// TwinCAT 3 PLC project kallebol_PLC_proj
// ProgramVersion: 3.1.4024.0
// libraries:
//   Tc2_MC2, * (Beckhoff Automation GmbH)
//   Tc2_Standard, * (Beckhoff Automation GmbH)
//   Tc2_System, * (Beckhoff Automation GmbH)
//   Tc3_Module, * (Beckhoff Automation GmbH)
// project tree:
//   / PlcTask.TcTTO
//   POUs/ MAIN.TcPOU
//   POUs/POUs/ FB_Azimuth.TcPOU, FB_Elevation.TcPOU
// real-time tasks:
//   TASK PlcTask: cycle T#10ms, priority 20, ADS port 350
// motion (NC):
//   TASK Azimuth_NC_task SAF: cycle T#2ms, priority 4, ADS port 501
//   TASK Azimuth_NC_task SVB: cycle T#10ms, priority 8, ADS port 511
//   AXIS Axis 3 (id 3)
//     General: UnitName=°
//     Dynamic: Acceleration=15000, Deceleration=15000, Jerk=64125
//     Velo: RefSearch=142.5, RefSync=142.5, SlowManual=712.5, FastManual=4275, Fast=14250, Maximum=14250
//     PositionAreaControl: Enable=false
//     TargetPosControl: Enable=false
//     OtherSettings: AllowMotionCmdToSlave=true
//     encoder EncType=8
//       EncPara: ScaleFactorNumerator=360, ScaleFactorDenominator=1048576, MaxCount=#xffffffff, EncPositionSource=1
//     drive DrvType=9
//       DrvPara: MaxCount=#xffffffff, DriveControlDWord=#x00030100
//         Analog: VeloReferenz=15675, VeloScale=1.02400649589962, TorqueSetpointScale=10, ScaleFactorActTorque=0.1
//         TimeComp: TaskDelayCycles=1
//     controller CtrType=1
//       CtrPara: PriorControlFactor=1
//         PosDiffControl: Enable=false
//         Observer: BandWidth=20
// I/O:
//   DEVICE Device 1 (EtherCAT), AmsNetId 5.79.241.154.2.1
//     Term 1 (EK1200) [EK1200-5000 EtherCAT Power supply (2A E-Bus)]
//       Term 2 (EL7342) [EL7342 2Ch. DC motor output stage (50V, 3.5A)]
//       RS485_term [EL6021 Interface (RS422/485)]
//       Term 3 (EK1110) [EK1110 EtherCAT extension]
//     Drive 4 (AX5203-0000-0214) [AX5203-0000-0214 EtherCAT Drive (SoE, 2 Ch.)]
// variable links:
//   Azimuth_NC_task SAF/Axes/Axis 3 <-> Device 1 (EtherCAT)/Drive 4 (AX5203-0000-0214)
//     Drive/Inputs/In/nDataIn1 <-> AT 1/Following distance
//     Drive/Inputs/In/nDataIn3[0] <-> AT 1/Torque/force feedback value
//     Drive/Inputs/In/nDcOutputTime <-> InfoData/DcOutputShift
//     Drive/Inputs/In/nState1 <-> AT 1/Drive status word @bit 8
//     Drive/Inputs/In/nState2 <-> AT 1/Drive status word
//     Drive/Inputs/In/nState4 @bit 1 <-> WcState/InputToggle
//     Drive/Inputs/In/nState4 <-> WcState/WcState
//     Drive/Outputs/Out/nCtrl1 <-> MDT 1/Master control word @bit 8
//     Drive/Outputs/Out/nDataOut1 <-> MDT 1/Position command value
//     Enc/Inputs/In/nDataIn1 <-> AT 1/Position feedback 1 value
//     Enc/Inputs/In/nDcInputTime <-> InfoData/DcInputShift
//     Enc/Inputs/In/nState4 @bit 1 <-> WcState/InputToggle
//     Enc/Inputs/In/nState4 <-> WcState/WcState
//   kallebol_PLC_proj/kallebol_PLC_proj Instance <-> Device 1 (EtherCAT)/Term 1 (EK1200)/Term 2 (EL7342)
//     PlcTask Inputs/MAIN.Elevation.Encoder_Value <-> ENC Status Channel 1/Counter value
//     PlcTask Inputs/MAIN.Elevation.Error <-> DCM Status Channel 1/Status/Error
//     PlcTask Inputs/MAIN.Elevation.Homing_Switch <-> DCM Status Channel 1/Status/Digital input 1
//     PlcTask Inputs/MAIN.Elevation.Limit_Switch <-> DCM Status Channel 1/Status/Digital input 2
//     PlcTask Inputs/MAIN.Elevation.Moving_negative <-> DCM Status Channel 1/Status/Moving negative
//     PlcTask Inputs/MAIN.Elevation.Moving_positive <-> DCM Status Channel 1/Status/Moving positive
//     PlcTask Inputs/MAIN.Elevation.Ready <-> DCM Status Channel 1/Status/Ready
//     PlcTask Inputs/MAIN.Elevation.Warning <-> DCM Status Channel 1/Status/Warning
//     PlcTask Outputs/MAIN.Elevation.Enable <-> DCM Control Channel 1/Control/Enable
//     PlcTask Outputs/MAIN.Elevation.Encoder_Setvalue <-> ENC Control Channel 1/Set counter value
//     PlcTask Outputs/MAIN.Elevation.Reset <-> DCM Control Channel 1/Control/Reset
//     PlcTask Outputs/MAIN.Elevation.Set_Encoder <-> ENC Control Channel 1/Control/Set counter
//     PlcTask Outputs/MAIN.Elevation.Target_Position <-> DCM Position Channel 1/Position
//   kallebol_PLC_proj/kallebol_PLC_proj Instance <-> Azimuth_NC_task SAF/Axes/Axis 3
//     PlcTask Inputs/MAIN.Azimuth.Azimuth_axis.NcToPlc <-> Outputs/ToPlc
//     PlcTask Outputs/MAIN.Azimuth.Azimuth_axis.PlcToNc <-> Inputs/FromPlc

CONFIGURATION kallebol_PLC_proj
    RESOURCE PLC ON TwinCAT3
        TASK PlcTask(INTERVAL := T#10ms, PRIORITY := 20);
        PROGRAM MAIN WITH PlcTask : MAIN;
    END_RESOURCE
END_CONFIGURATION

// ---- POUs/MAIN.TcPOU
PROGRAM MAIN
VAR
Elevation : FB_Elevation;
Azimuth : FB_Azimuth;
END_VAR

Elevation();
Azimuth();

END_PROGRAM

// ---- POUs/POUs/FB_Elevation.TcPOU
FUNCTION_BLOCK FB_Elevation
VAR_INPUT
END_VAR
VAR_OUTPUT
END_VAR
VAR
	
	//Data for ADS communtication
	Targetpos_mm 			: LREAL	:= 0;		//Data FROM ADS
	Targetpos_deg			: LREAL := 0;		//Data FROM ADS
	Current_Position_mm 	: LREAL;			//Data TO ADS
	Current_Position_deg 	: LREAL; 			//Data from inclonometer, updated asynchronous from RS485
	Enable AT %Q* 			: BOOL 	:= FALSE;	//Data FROM ADS
	Homeing 				: BOOL 	:= FALSE;	//Data TO ADS
	Homeing_Error 			: BOOL 	:= FALSE;	//Data TO ADS
	Homeing_Wrong_direction : BOOL  := FALSE;	//Data TO ADS
	Reset_requested 		: BOOL  := FALSE;	//Data FROM ADS
	Error AT %I* 			: BOOL;				//Data TO ADS
	Target_in_deg			: BOOL  := FALSE;	//DATA FROM ADS
	//Position_Error AT %I* 	: BOOL;
	
		
	//Data for ADS communtication END
	
	
	Reset AT %Q* 			: BOOL 	:= FALSE;
	Encoder_Value AT %I* : UDINT;
	Homing_Switch AT %I* : BOOL;
	Limit_Switch AT %I* : BOOL;
	Warning AT %I* : BOOL;

	Ready AT %I* : BOOL;
	Moving_positive AT %I* : BOOL;
	Moving_negative AT %I* : BOOL;
	//In_target AT %I* : BOOL;
	Set_Encoder AT %Q* : BOOL;
	Encoder_Setvalue AT %Q* : UDINT;
	Target_Position AT %Q* : UDINT;
	
	P_error : LREAL; //position error
	Ang_P_fac : REAL := 0.01; //This is not really a P factor, I think it's more of a I
 	//Ang_I_fac : REAL := 0.001;


	Homed : BOOL := FALSE;
	Homeing_Allowed : BOOL := TRUE;
	Homeing_State : UINT := 0;
	Reset_state : UINT := 0;
	
	Homeing_check_home_direction : BOOL := TRUE; //If we want to check weather the homeing is in the correct direction
	Homeing_debouceing_home_switch : BOOL := FALSE; //Used to debouce 
	Homing_started_mm : LREAL; // to monitor if the homeing goes the right direction
	
	Homeing_Timer : TON; //used for timeouts
	Homeing_Timer2 : TON;
	
	
	
END_VAR

VAR CONSTANT
	maxmove_mm : LREAL := 210;
	minmove_mm : LREAL := 0;
	Zeroposition : UDINT := 1000000;
END_VAR

IF Homeing_Error THEN
	enable := FALSE;
	Homeing_state := 0;
	Homed := FALSE;
END_IF

IF Reset_requested THEN
	Reset_Elevation();
END_IF

IF Homed = FALSE AND Enable = TRUE AND Homeing_Allowed AND Homeing_Error = FALSE THEN
	//The homing sequence should start automaticly if the PLC is restarted and Enable is set
	Homeing_sequence();
ELSE
	IF Homed = TRUE AND Enable = TRUE THEN //Normal operation
		IF Target_in_deg = FALSE THEN
			//'Dumb' positioning, semi-openloop the position is only based on the 
			//Encoder value, not the actual measured value
			Target_Position := mm_to_encoder(LIMIT(minmove_mm,targetpos_mm,maxmove_mm));
		ELSE
			//closed-loop positionin with a inclonometer in the loop
			//Requires that the inclonometer is working
			P_error := Current_Position_deg - Targetpos_deg;
			Target_Position := mm_to_encoder(LIMIT(minmove_mm,
			Target_Position + P_error*Ang_P_fac
			,maxmove_mm));
		END_IF
	
	
		
	END_IF
END_IF

current_position_mm := encoder_to_mm(Encoder_Value);

METHOD encoder_to_mm : LREAL
VAR_INPUT
	encoder_pos : UDINT;
END_VAR

VAR
	encoder_ppr : LREAL := 2000;
	mm_per_rev : LREAL := 0.8; //calibrate this value
END_VAR
encoder_to_mm := UDINT_TO_LREAL(encoder_pos - Zeroposition) / (encoder_ppr * mm_per_rev);
END_METHOD

METHOD Homeing_sequence : BOOL
VAR_INPUT
END_VAR
VAR
	diff_pos : LREAL;
END_VAR
Homeing_Timer(IN:=TRUE, PT:= T#200S); //timeout of the homeing, it takes a long time to home...
Homeing := TRUE;

IF Homeing_Timer.Q THEN
	//Timeout as been reached
	Homeing_Error := TRUE;
	Homeing_Timer(IN:=FALSE);
END_IF

IF Homing_Switch AND Homeing_state < 3 THEN
	IF Homeing_debouceing_home_switch THEN
		Homeing_state := 3;
	END_IF
	Homeing_debouceing_home_switch := TRUE;
ELSE
	Homeing_debouceing_home_switch := FALSE; //There is some weird stuff with the homeswitch some times, maybe we are using the DYN output of the ABB EDEN switch?
END_IF

CASE Homeing_state OF
	0:
	 	//We want to set the current position to a high number so we can go into the negative as the countervalue is a UDINT
		Encoder_Setvalue := Zeroposition;
		Target_Position  := Zeroposition;
		Set_Encoder := 1;
		Homeing_Timer2(IN:= TRUE, PT:= T#1S);
		IF Homeing_Timer2.Q THEN
			Homeing_Timer2(IN:=FALSE);
			Homeing_state := 1;
		END_IF
			
	1:
		Set_Encoder := 0;
		
		Homeing_Timer2(IN:= TRUE, PT:= T#1S);
		IF Homeing_Timer2.Q THEN
			Homeing_Timer2(IN:=FALSE);
			Homeing_state := 2;
			Homing_started_mm := encoder_to_mm(Encoder_Value);
		END_IF
	2: 
		//Goes to a position in the 'negatives' 
		Target_Position := 0;
		diff_pos := (encoder_to_mm(Encoder_Value) - Homing_started_mm);
		//Diff_pos will be very large if it is going the correct direction due to underflow
		//If it does not grow large, it is going the wrong way 
		IF Homeing_check_home_direction AND diff_pos > 10 AND diff_pos < 1000 THEN
			// for some reason this happens sometime
			homeing_error := TRUE;
			Homeing_Wrong_direction := TRUE;
		END_IF
		
	3: 
		//The limit switch has been reached
		//Stop the motor and set the new zero when the motor has stopped
		Target_Position := Encoder_Value; //Stop the motor without disabling it
		Homeing_Timer2(IN:= TRUE, PT:= T#2S);
		//A small delay to allow the motor to stabilize
		IF Homeing_Timer2.Q THEN
			Encoder_Setvalue := Zeroposition;
			Target_Position := Zeroposition;
			Set_Encoder := 1;
			Homeing_state := 4;
			Homeing_Timer2(IN:=FALSE);
		END_IF
		
	4: 
	
		//Motor has been homed
		Set_Encoder := 0;
		Homeing_Timer(IN:=FALSE);
		Homeing := FALSE;
		Homed := TRUE;
		homeing_state := 0;
		
	
END_CASE
END_METHOD

METHOD mm_to_encoder : UDINT
VAR_INPUT
	mm_in : LREAL;
END_VAR
VAR
	encoder_ppr : LREAL := 2000;
	mm_per_rev : LREAL := 0.8; //calibrate this value
END_VAR
mm_to_encoder := LREAL_TO_UDINT(mm_in* mm_per_rev * encoder_ppr) + Zeroposition;
END_METHOD

METHOD Reset_Elevation : BOOL
VAR_INPUT
END_VAR

CASE Reset_state OF
	0:
		enable := FALSE;
		Reset_state := 1;
	1:
		Reset := TRUE;
		Targetpos_mm := Current_Position_mm ;
		Homed := FALSE;
		Homeing_Error := FALSE;
		Homeing_Wrong_direction := FALSE;
		Homeing_State := 0;
		Reset_state := 2;
		
	2: 
		Reset := FALSE;
		Reset_state := 3;
		
	3: //A extra one for good luck
		Reset := TRUE;
		Reset_state := 3;
		
	4: 
		Reset := FALSE;
		Reset_state := 0;
		Reset_requested := FALSE;
	
END_CASE
END_METHOD

METHOD set_Current_Position_deg : BOOL
VAR_INPUT
	deg : LREAL;
END_VAR
Current_Position_deg := deg;
END_METHOD

END_FUNCTION_BLOCK

// ---- POUs/POUs/FB_Azimuth.TcPOU
FUNCTION_BLOCK FB_Azimuth
VAR
	
	EnableAzimuth : BOOL := FALSE; //For ADS


	Azimuth_Target_Position_Parabola : LREAL := 0; // for ADS, target position in 'real' angles
	HMI_Azimuth : LREAL; //Readable position, scaled for your pleasure for ADS
	
	Azimuth_target_position : LREAL := 0; //in motor angles, 
	
	Azimuth_CurrentPosition : LREAL;
	Azimuth_Old_position : LREAL;
	Azimuth_Moveto_position :LREAL;
	Azimuth_state : INT := 1;
	Azimuth_enable_tracking : BOOL := FALSE;
	Azimuth_setpoint_scaled: REAL;
	Azimuth_actual_position : LREAL;
	
	Azimuth_axis : AXIS_REF; 
	Azimuth_PowerAxis: MC_Power;
	Azimuth_PowerAxisOut: ST_McOutputs;
	Azimuth_MoveAxis: MC_MoveAbsolute;
	Azimuth_MoveAbsoluteOut: ST_McOutputs;
	Azimuth_ResetOut: ST_McOutputs;
	

	Azimuth_Axis_power : MC_Power;
	Azimuth_axis_move_abs : MC_moveAbsolute;
	Azimuth_Reset : MC_Reset;
	
	Azimuth_timer : TON; //Timer for init of Azimuth_axis
END_VAR

VAR CONSTANT
	Azimuth_zero : REAL := 0; //'fake' zero position
	Gearratio : REAL := 0.0011904761904762;//1.0/840.0;

END_VAR


IF EnableAzimuth = FALSE THEN
	Azimuth_state := 0;
END_IF

IF EnableAzimuth = TRUE AND Azimuth_state = 0 THEN
	Azimuth_state := 1;
END_IF
 
 update_Azimuth();

METHOD update_Azimuth : BOOL
VAR_INPUT
END_VAR
VAR CONSTANT
	Invert_Azimuth_axis : BOOL := FALSE;
END_VAR
Azimuth_axis();

Azimuth_target_position := Azimuth_Target_Position_Parabola/gearratio;

IF Invert_Azimuth_axis THEN
	Azimuth_setpoint_scaled := LREAL_TO_REAL(Azimuth_target_position);
	Azimuth_CurrentPosition := LREAL_TO_REAL(Azimuth_axis.NcToPlc.ActPos);
	Azimuth_actual_position := LREAL_TO_REAL(Azimuth_axis.NcToPlc.ActPos - Azimuth_zero);
	
	Azimuth_Moveto_position := Azimuth_zero + Azimuth_target_position; 
ELSE
	Azimuth_setpoint_scaled := LREAL_TO_REAL(Azimuth_target_position);
	Azimuth_CurrentPosition := Azimuth_axis.NcToPlc.ActPos;
	Azimuth_actual_position := Azimuth_zero - Azimuth_axis.NcToPlc.ActPos;
	
	Azimuth_Moveto_position := Azimuth_zero - Azimuth_target_position; 

END_IF
CASE Azimuth_state OF
	-1 : //Error state
			IF Azimuth_axis.Status.Error THEN
				Azimuth_state := 4;	(* axis error requires reset *)
			ELSE
				Azimuth_state := 1;	(* function block errors don't need a reset *)
			END_IF
		
	0 : //Stopped
			Azimuth_MoveAxis.Execute := FALSE;
			Azimuth_PowerAxis.Enable := FALSE;
			Azimuth_PowerAxis.Enable_Positive := FALSE;
			Azimuth_PowerAxis.Enable_Negative := FALSE;
	1 : //INIT
			Azimuth_MoveAxis.Execute := FALSE;
			Azimuth_Reset.Execute := FALSE;
			Azimuth_state := 2;	
			IF Azimuth_PowerAxis.Error THEN
				Azimuth_state := -1;
			END_IF
	2 : //Enabled but not moving
			Azimuth_PowerAxis.Enable := TRUE;
			Azimuth_PowerAxis.Enable_Positive := TRUE;
			Azimuth_PowerAxis.Enable_Negative := TRUE;
			Azimuth_MoveAxis.BufferMode := MC_aborting;
			IF EnableAzimuth AND Azimuth_axis.Status.Operational THEN
				Azimuth_state := 33;
				Azimuth_enable_tracking := TRUE;
			END_IF
			
			IF Azimuth_PowerAxis.Error THEN
				Azimuth_state := -1;
			END_IF
	
	33 : //Tracking mode, tries to follow Azimuth value 

		
			//Pulse .Execute since movement is triggered on rising edge
			IF Azimuth_MoveAxis.Execute THEN
				Azimuth_MoveAxis.Execute := FALSE;
			ELSE
				//IF movements are large enough
				IF ABS(Azimuth_Moveto_position - Azimuth_axis.NcToPlc.ActPos) > 0.04 OR ABS(Azimuth_Moveto_position - Azimuth_Old_position) > 0.04 THEN
					Azimuth_Old_position := Azimuth_Moveto_position;
					Azimuth_MoveAxis.Position := Azimuth_Moveto_position;
					Azimuth_MoveAxis.Acceleration  := 40_000;
					Azimuth_MoveAxis.Deceleration  := 40_000;
					Azimuth_MoveAxis.Jerk 			:= 10_000;
					Azimuth_MoveAxis.Velocity 		:= 14000;

					Azimuth_MoveAxis.Execute 		:= TRUE;
					
				ELSE
					Azimuth_MoveAxis.Execute := FALSE;
				END_IF
			END_IF

			IF Azimuth_enable_tracking = FALSE THEN //If tracking is no longer desired
				Azimuth_state := 2;
			END_IF
			IF Azimuth_MoveAxis.CommandAborted OR Azimuth_MoveAxis.Error OR Azimuth_axis.Status.Error THEN //Machine error
				Azimuth_state := -1;
			END_IF
			
	4: //Reset
			Azimuth_Reset.Execute := TRUE;
			IF Azimuth_Reset.Done THEN
				Azimuth_state := 1;
			ELSIF Azimuth_Reset.Error THEN
				Azimuth_state := 1; 
			END_IF

END_CASE


IF Invert_Azimuth_axis THEN
	HMI_Azimuth := Azimuth_axis.NcToPlc.ActPos*gearratio - Azimuth_zero;
ELSE
	HMI_Azimuth := Azimuth_zero - Azimuth_axis.NcToPlc.ActPos*gearratio;

END_IF

Azimuth_Axis_power(		
	Axis:=Azimuth_axis,
	Enable:=Azimuth_PowerAxis.Enable,
	Enable_positive:=Azimuth_PowerAxis.Enable_Positive,
	Enable_negative:=Azimuth_PowerAxis.Enable_Negative,
	Override:=100,
	Status =>Azimuth_PowerAxisOut.done,
	Busy=>Azimuth_PowerAxisOut.Busy,
	Active=>Azimuth_PowerAxisOut.Active,
	Error=>Azimuth_PowerAxisOut.Error,
	ErrorID => Azimuth_PowerAxisOut.ErrorID
);

Azimuth_axis_move_abs(
	Axis:=Azimuth_axis,
	execute:=Azimuth_MoveAxis.Execute,
	Position:=Azimuth_MoveAxis.Position,
	Velocity:=Azimuth_MoveAxis.Velocity,
	Acceleration:=Azimuth_MoveAxis.Acceleration,
	Deceleration:=Azimuth_MoveAxis.Deceleration,
	BufferMode:=Azimuth_MoveAxis.BufferMode,
	Jerk:=Azimuth_MoveAxis.Jerk,
	Done=>Azimuth_MoveAbsoluteOut.Done,
	Busy=>Azimuth_MoveAbsoluteOut.Busy,
	Active=>Azimuth_MoveAbsoluteOut.Active,
	CommandAborted=>Azimuth_MoveAbsoluteOut.CommandAborted,
	Error=>Azimuth_MoveAbsoluteOut.Error,
	ErrorID=>Azimuth_MoveAbsoluteOut.ErrorID
);

Azimuth_Reset(
	Axis:=Azimuth_axis,
	Execute:=Azimuth_Reset.Execute,
	Busy=>Azimuth_ResetOut.Busy,
	Error=>Azimuth_ResetOut.Error,
	ErrorID=>Azimuth_ResetOut.ErrorID
);
END_METHOD

END_FUNCTION_BLOCK
